Fanuc KAREL source: kb00135.KL

-- PROVISIONAL review KL for V940-1; original PC SHA256 f07a18ea391237f31418e81f8ab9ba24a701a1281175b499900c305da66ff03d
-- Incomplete behavior may be omitted. Consult companion uncertainty JSON. Do not deploy.
PROGRAM KB00135
%NOLOCKGROUP
BEGIN
  -- V9_ZERO_TABLE_METADATA_HINT layout=0002_ascii; no indexed target words; source/name/runtime held
  -- UNRESOLVED_PC offsets 5-12; opcodes 9D,23
  -- UNRESOLVED_PC offsets 17-26; opcodes 3F,75
  -- UNRESOLVED_PC offsets 31-38; opcodes 9D,23
  -- UNRESOLVED_PC offsets 43-50; opcodes 9D,23
  -- UNRESOLVED_PC offsets 55-85; opcodes 27,22,22,2A,22,22,31
  -- UNRESOLVED_PC offsets 90-94; opcodes 7F
END KB00135
